Universal Robots PolyScope program: accept_order.urp

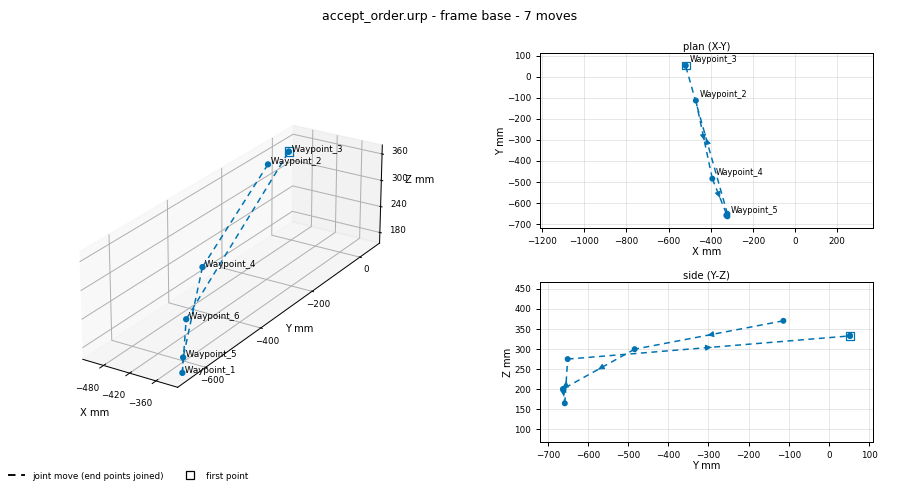
[picture p0: tool path of accept_order.urp in frame base, 7 of 8 moves have a stored position in this frame; points joined in program order, loops and branches not executed]
Program accept_order (installation=default directory=/programs/AronLauschOrdering createdIn=5.9.5.1031259 lastSavedIn=5.12.6.1102099 robotSerialNumber=20215500597)
Calibrated DH parameters: a=[0.000193, -0.066673, -0.391568, -0.000012, 0.00005, 0]; d=[0.162643, -472.05677, 465.132521, 7.058239, 0.099746, 0.099582]; alpha=[1.571116, 0.00089, 0.003862, 1.569269, -1.569248, 0]; deltaTheta=[0, -1.413394, 7.628392, 0.068187, 0, -0.000001]
Robot Program (runOnlyOnce=true)
  MoveJ speed 60 deg/s, acceleration 80 deg/s^2 (useActiveTCP=true) feature=Base
    Waypoint Waypoint_3: TCP in base x=-519.145 y=52.76 z=332.958 mm, rx=-3.1405 ry=-0.0837 rz=0.0002 rad; joints [-20.664, -88.123, 82.733, -84.528, -89.812, 66.326] deg; TCP offset x=0 y=0 z=191.5 mm, rx=0 ry=0 rz=0 rad
    URCap Gripper (Robotiq_Grippers, Robotiq Inc.) dataModel(position=0.0, force=100.0, speed=100.0, positionInDouble=0.0, forceInDouble=100.0, speedInDouble=100.0, slaveIds=[9], blocking=true)
    URCap Gripper Activate (Robotiq_Grippers, Robotiq Inc.) dataModel(ResetAndActivateKey=false)
  order_plattform := [GP_int_in[0]]
  MoveJ speed 60 deg/s, acceleration 80 deg/s^2 (useActiveTCP=true) feature=Base
    offset_pos := p[-0.12*order_plattform[0],0,0,0,0,0]
    glass_selected := pose_add(firstscale,offset_pos)
    Waypoint Waypoint (Variable): variable(name=glass_selected)
  MoveL speed 250 mm/s, acceleration 1200 mm/s^2 (useActiveTCP=true) feature=Base
    MoveDirectionNode (selectedDirection=ZMinus)
      Until DISTANCE (allowActions=false deceleration=3 distanceNodeType=STOP) Distance=0.05; motionParameters(blendRadius=0)
    URCap Gripper (Robotiq_Grippers, Robotiq Inc.) dataModel(position=100.0, force=60.0, speed=100.0, positionInDouble=100.0, forceInDouble=60.0, speedInDouble=100.0, slaveIds=[9], blocking=true)
    MoveDirectionNode (selectedDirection=ZPlus)
      Until DISTANCE (allowActions=false deceleration=3 distanceNodeType=STOP) Distance=0.06; motionParameters(blendRadius=0)
  MoveJ speed 60 deg/s, acceleration 80 deg/s^2 (useActiveTCP=true) feature=Base
    Waypoint Waypoint_2: TCP in base x=-470.319 y=-113.347 z=370.532 mm, rx=3.078 ry=0.6285 rz=0 rad; joints [-2.507, -92.708, 81.739, -78.942, -89.816, 64.437] deg
    Waypoint Waypoint_4: TCP in base x=-392.295 y=-483.981 z=299.838 mm, rx=-2.6646 ry=-1.6641 rz=0.0001 rad; joints [38.579, -74.057, 71.151, -87.009, -89.812, 64.648] deg
    Waypoint Waypoint_5: TCP in base x=-320.581 y=-662.671 z=200.67 mm, rx=-3.1402 ry=-0.0898 rz=-0.0001 rad; joints [53.721, -56.831, 60.673, -93.747, -89.799, 140.497] deg; TCP offset x=0 y=0 z=191.5 mm, rx=0 ry=0 rz=0 rad
    Waypoint Waypoint_1: TCP in base x=-325.774 y=-658.115 z=164.889 mm, rx=-3.1407 ry=-0.0744 rz=0 rad; joints [53.172, -56.504, 65.409, -98.814, -89.8, 140.53] deg; TCP offset x=0 y=0 z=191.5 mm, rx=0 ry=0 rz=0 rad
    URCap Gripper (Robotiq_Grippers, Robotiq Inc.) dataModel(position=0.0, force=100.0, speed=100.0, positionInDouble=0.0, forceInDouble=100.0, speedInDouble=100.0, slaveIds=[9], blocking=true)
    Waypoint Waypoint_6: TCP in base x=-320.589 y=-650.963 z=275.149 mm, rx=3.1407 ry=0.0713 rz=-0.0001 rad; joints [53.171, -58.337, 52.17, -83.749, -89.803, 140.584] deg
    Waypoint Waypoint_3: TCP in base x=-519.145 y=52.76 z=332.958 mm, rx=-3.1405 ry=-0.0837 rz=0.0002 rad; joints [-20.664, -88.123, 82.733, -84.528, -89.812, 66.326] deg
